PROGRAM MAIN
VAR
	brun 		AT %Q* : BOOL;
	bACK 		AT %Q* : BOOL;
	bSafety_OK  AT %I* : BOOL;
	bInit              : BOOL;
	Initialize		   : R_TRIG;
	Ack_Input		   : BOOL;
	Safety_Timer       : TON;	
	SafeOP_Timer	   : TON;
	EMG_Raise		   : R_TRIG;
	OP10A_Robo_State AT %I* : USINT;
	OP10B_Robo_State AT %I* : USINT;

	SERVO_TORQUE	AT %Q*	:UINT := 10000;
	
	ALL_LIGHTS_ON: BOOL;
	XTS_Lube_ON  : BOOL;
	
	All_Station_Auto_Mode     : BOOL;
	All_Station_Cycle_Start   : BOOL;
	All_Station_Cycle_Stop    : BOOL;
	Station_Ctrl_Temp         : BOOL;
	OP10_Lights_On			  : BOOL;
	tower_lamp_green_on       :BOOL;
	tower_lamp_red_on         :BOOL;
	tower_lamp_orange_on: BOOL;
	
	FB_Timer : FB_Time_Stamp_Maddy;
	Run_Time : STRING;
	Start_timer : BOOL;
	Stop_timer  : BOOL;
	Reset_timer : BOOL;
	Start_value : STRING;
	Stop_value  : STRING;
	Start_trig : R_TRIG;
	Stop_Trig  : R_TRIG;
	Reset_Trig : R_TRIG;
END_VAR


bACK			:= Pulse_Block.Q1Hz;

//Axis_Position_Bias();
O160_AUTOBAG_CNT_CMPLTD_Q707_4:=I10A_DRUM_OFF_ON_I714_2;
Initialize(CLK:=NOT bInit);
IF Initialize.Q THEN
	Ack_Input:=1;
	brun:=TRUE;
END_IF
SafeOP_Timer(IN:=Ack_Input,PT:=T#5S);
IF SafeOP_Timer.Q THEN
 bACK:=TRUE;
 Ack_Input:=0;
 bInit:=TRUE;
END_IF

Safety_Timer(IN:=bACK,PT:=T#500MS);
IF Safety_Timer.Q THEN
	bACK:=FALSE;
END_IF

EMG_Raise(CLK:=bSafety_OK , Q=> );
IF EMG_Raise.Q THEN
   bACK:=TRUE;
END_IF

RFID();
Error();
OP10_MAIN();
OP20_MAIN();
OP30_MAIN();
OP40_MAIN();
OP50_MAIN();
OP60_MAIN();
OP70_MAIN();
OP80_MAIN();
OP90_MAIN();
OP110_MAIN();
OP120_MAIN();
OP130_MAIN();
OP140_MAIN();
OP160_MAIN();
IO_Diag();
IO_OP10_PANEL();
IO_OP10A_10B_JB();
Master1_IO_Map();
MASTER2_IO_Map();
OP90_MP_IO();
OP90_MASTER3_IO();
OP90_JB_IO();
OP160_MP_IO();
OP160_MASTER4_IO();
OP120_JB_IO();
OP150_Main();
MAIN_1();
EtherCatDiag();
//MOdeselection From HMI
IF (HMI_AutoMode AND NOT HMI_ManualMOde AND NOT HMI_StepMode) THEN
		FB_MODE_BLOCK.ModeWord:=1;
	ELSIF (NOT HMI_AutoMode AND HMI_ManualMOde AND NOT HMI_StepMode) THEN
		FB_MODE_BLOCK.ModeWord:=2;
	ELSIF  (NOT HMI_AutoMode AND NOT HMI_ManualMOde AND HMI_StepMode) THEN
		FB_MODE_BLOCK.ModeWord:=3;
    ELSE   
		FB_MODE_BLOCK.ModeWord:=0;
END_IF

Servo_safety     := bSafety_OK;
OperationEnable  := bSafety_OK;

IF OperationEnable THEN
	Servo_Enable:=TRUE;
ELSE
	Servo_Enable:=FALSE;
END_IF

FB_MODE_BLOCK(
	ModeWord:= , 
	HomeConditionOK:= ALL_STN_IN_HOME, 
	OperationEnable:= bSafety_OK , 
	StartPB:= START_PB, 
	SafetyAndNOError:= bSafety_OK AND NOT ERROR_ACTIVE, 
	ModeAck:= TRUE , 
	HomingINProgress:= , 
	TempHomeOK:= , 
	ResetPB:= , 
	AutoSelected=>AUTO_SELECTED , 
	ManualSelected=> MANUAL_SELECTED, 
	StepSelected=> STEP_SELECTED, 
	ModeSelAck_Indication=> , 
	StatusDisplay=> , 
	AutoRunning:=AUTO_RUNNING , 
	StepRunning:=STEP_RUNNING , 
	StartEnable:=START_ENABLE , 
	MachineStop:=MACHINE_STOP);
	
Pulse_Block(
	Q10Hz=> , 
	Q5Hz=> , 
	Q2_5Hz=> , 
	Q2Hz=> , 
	Q1_25Hz=> , 
	Q2Hz=> , 
	Q0_625Hz=> , 
	Q0_5Hz=> );	
	
IF ALL_LIGHTS_ON THEN				
		O30_CAM_LGHT1_ON_Q305_1                  :=1;
		O30_CAM_LGHT2_ON_Q305_2                  :=1;
		O50_CAM_LGHT1_ON_Q306_3                  :=1;
		O50_CAM_LGHT2_ON_Q306_4                  :=1;
		O70_CAM_LGHT1_ON_Q307_6                  :=1;
		O70_CAM_LGHT2_ON_Q307_7                  :=1;
		O90_VISN_LGHT1_ON_Q400_0                 :=1;
		O90_VISN_LGHT2_ON_Q400_1                 :=1;
		O120_VISN_LGHT1_ON_Q402_4                :=1;
		O120_VISN_LGHT2_ON_Q402_5                :=1;
		O150_VISN_LGHT_ON_Q706_6                 :=1;
		O160_CHECKER_LGHT_ON_Q707_1              :=1;
ELSE		
		O30_CAM_LGHT1_ON_Q305_1                  :=0;
		O30_CAM_LGHT2_ON_Q305_2                  :=0;
		O50_CAM_LGHT1_ON_Q306_3                  :=0;
		O50_CAM_LGHT2_ON_Q306_4                  :=0;
		O70_CAM_LGHT1_ON_Q307_6                  :=0;
		O70_CAM_LGHT2_ON_Q307_7                  :=0;
		O90_VISN_LGHT1_ON_Q400_0                 :=0;
		O90_VISN_LGHT2_ON_Q400_1                 :=0;
		O120_VISN_LGHT1_ON_Q402_4                :=0;
		O120_VISN_LGHT2_ON_Q402_5                :=0;
		O150_VISN_LGHT_ON_Q706_6                 :=0;
		O160_CHECKER_LGHT_ON_Q707_1              :=0;	
END_IF

IF OP10_Lights_On THEN
		O10A_BDY_EMPT_CAM_LGHT1_ON_Q301_0        :=1; 
		O10A_BDY_EMPT_CAM_LGHT2_ON_Q301_1        :=1;
//		O10A_FIRTREE_ORING_CAM_LGHT1_ON_Q301_2   :=1;
//		O10A_FIRTREE_ORING_CAM_LGHT2_ON_Q301_3   :=1;
		O10A_ORING_CAM_LGHT1_ON_Q301_4           :=1;
		O10A_ORING_CAM_LGHT2_ON_Q301_5           :=1;
//		O10A_FIRTREE_ORING_CAMBAR_LGHT1_ON_Q301_6:=1;
//		O10B_FIRTREE_ORING_CAM_LGHT1_ON_Q303_2   :=1;
//		O10B_FIRTREE_ORING_CAM_LGHT2_ON_Q303_3   :=1;
		O10B_ORING_CAM_LGHT1_ON_Q303_4           :=1;
		O10B_ORING_CAM_LGHT2_ON_Q303_5           :=1;
//		O10B_FIRTREE_ORING_CAMBAR_LGHT1_ON_Q303_6:=1;
ELSE
		O10A_BDY_EMPT_CAM_LGHT1_ON_Q301_0        :=0; 
		O10A_BDY_EMPT_CAM_LGHT2_ON_Q301_1        :=0;
		O10A_FIRTREE_ORING_CAM_LGHT1_ON_Q301_2   :=0;
		O10A_FIRTREE_ORING_CAM_LGHT2_ON_Q301_3   :=0;
		O10A_ORING_CAM_LGHT1_ON_Q301_4           :=0;
		O10A_ORING_CAM_LGHT2_ON_Q301_5           :=0;
		O10A_FIRTREE_ORING_CAMBAR_LGHT1_ON_Q301_6:=0;
		O10B_FIRTREE_ORING_CAM_LGHT1_ON_Q303_2   :=0;
		O10B_FIRTREE_ORING_CAM_LGHT2_ON_Q303_3   :=0;
		O10B_ORING_CAM_LGHT1_ON_Q303_4           :=0;
		O10B_ORING_CAM_LGHT2_ON_Q303_5           :=0;
		O10B_FIRTREE_ORING_CAMBAR_LGHT1_ON_Q303_6:=0;	
END_IF
		
		
IF XTS_Lube_ON THEN
	O10_XTS_GREASE_VALVE_ON_Q300_0:=Pulse_Block.Q0_5Hz;
ELSE	
	O10_XTS_GREASE_VALVE_ON_Q300_0:=0;
END_IF
		
O150_BARLIGHT_OP1_Q706_7 :=	Pulse_Block.Q2_5Hz;
O150_BARLIGHT_OP2_Q707_0 := Pulse_Block.Q1Hz;	
                                                      
O10_TWR_LMP_RD_Q302_5   := Pulse_Block.Q1Hz AND tower_lamp_green_on;                         
O10_TWR_LMP_GN_Q302_6   := Pulse_Block.Q1Hz AND tower_lamp_red_on;                        
O10_TWR_LMP_YELW_Q302_7 := Pulse_Block.Q1Hz AND tower_lamp_orange_on;
O120_TWR_LMP_GN_Q403_1   := Pulse_Block.Q1Hz AND tower_lamp_green_on;
O120_TWR_LMP_YELW_Q403_2 := Pulse_Block.Q1Hz AND tower_lamp_orange_on ;
O120_TWR_LMP_RD_Q403_0   := Pulse_Block.Q1Hz AND tower_lamp_red_on;	

O10_BARLIGHT_OP1_Q300_6  := Pulse_Block.Q1Hz;
O10_BARLIGHT_OP2_Q300_7  := Pulse_Block.Q1_25Hz;	

IF NOT OperationEnable THEN
	OP20_ErrorActive:=1;
	OP30_ErrorActive:=1;
	OP40_ErrorActive:=1;
	OP50_ErrorActive:=1;
	OP60_ErrorActive:=1;
	OP70_ErrorActive:=1;
	OP80_ErrorActive:=1;
	OP110_ErrorActive:=1;
	OP120_ErrorActive:=1;
	OP130_ErrorActive:=1;
	OP140_ErrorActive:=1;
	OP160_ErrorActive:=1;
END_IF

IF AUTO_WITH_XTS AND Station_Ctrl_Temp THEN

	IF All_Station_Auto_Mode THEN
		OP20_HMI_AutoMode:=1;
		OP30_HMI_AutoMode:=1;
		OP40_HMI_AutoMode:=1;
		OP50_HMI_AutoMode:=1;
		OP60_HMI_AutoMode:=1;
		OP70_HMI_AutoMode:=1;
		OP80_HMI_AutoMode:=1;	
		OP110_HMI_AutoMode:=1;	
        OP120_HMI_AutoMode:=1;
		OP130_HMI_AutoMode:=1;	
	//	OP140_HMI_AutoMode:=1;
        OP160_HMI_AutoMode:=1;			
	END_IF
	IF All_Station_Cycle_Start THEN
		OP20_HMI_CycleStart	:=1;
		OP30_HMI_Cycle_Start:=1;
		OP40_HMI_Cycle_Start:=1;
		OP50_HMI_Cycle_Start:=1;
		OP60_HMI_CycleStart	:=1;
		OP70_HMI_Cycle_Start:=1;
		OP80_HMI_CycleStart	:=1;
		OP110_HMI_CycleStart:=1;
		OP120_HMI_CycleStart_PB:=1;
		OP130_HMI_CycleStart:=1;
	//	OP140_HMI_CycleStart:=1;
		OP160_HMI_CycleStart:=1;
	ELSE
		OP20_HMI_CycleStart	:=0;
		OP30_HMI_Cycle_Start:=0;
		OP40_HMI_Cycle_Start:=0;
		OP50_HMI_Cycle_Start:=0;
		OP60_HMI_CycleStart	:=0;
		OP70_HMI_Cycle_Start:=0;
		OP80_HMI_CycleStart	:=0;
		OP110_HMI_CycleStart:=0;	
		OP120_HMI_CycleStart_PB:=0;
		OP130_HMI_CycleStart:=0;
	//	OP140_HMI_CycleStart:=0;
		OP160_HMI_CycleStart:=0;		
	END_IF
	IF All_Station_Cycle_Stop THEN
		 OP20_Stop_Request  :=1;
 		 OP30_Stop_Request  :=1;
 		 OP40_Stop_Request  :=1;
 		 OP50_Stop_Request  :=1;
 		 OP60_Stop_Request  :=1;
 		 OP70_Stop_Request  :=1;
 		 OP80_Stop_Request  :=1;
 		 OP110_Stop_Request :=1;
		 OP120_Machine_Stop :=1;
		 OP130_Machine_Stop	:=1;
		// OP140_Machine_Stop :=1;
		 OP160_Machine_Stop	:=1;
	ELSE
		 OP20_Stop_Request  :=0;
 		 OP30_Stop_Request  :=0;
 		 OP40_Stop_Request  :=0;
 		 OP50_Stop_Request  :=0;
 		 OP60_Stop_Request  :=0;
 		 OP70_Stop_Request  :=0;
 		 OP80_Stop_Request  :=0;
 		 OP110_Stop_Request :=0;
		 OP120_Machine_Stop :=0;
		 OP130_Machine_Stop	:=0;
		// OP140_Machine_Stop :=0;
		 OP160_Machine_Stop	:=0;	 
	END_IF
END_IF	


////// tower lamp ////////////////////
IF OP10A_AUTO_RUNNING AND  OP160_AutoRunning AND  OP140_AutoRunning AND 
   OP130_AutoRunning AND OP110_AutoRunning AND OP120_AutoRunning  AND 
   OP90_AUTO_RUNNING AND OP80_AutoRunning AND OP70_AutoRunning AND 
   OP60_AutoRunning AND  OP50_AutoRunning AND OP40_AutoRunning AND 
   OP30_AutoRunning AND OP20_AutoRunning THEN
   tower_lamp_green_on := TRUE;
   tower_lamp_red_on   := FALSE;
   tower_lamp_orange_on:=FALSE;	
END_IF

IF NOT (OP160_AutoRunning AND  OP140_AutoRunning AND  OP130_AutoRunning AND 
        OP10A_AUTO_RUNNING AND OP110_AutoRunning AND OP120_AutoRunning AND
        OP90_AUTO_RUNNING AND OP80_AutoRunning AND OP70_AutoRunning AND
        OP60_AutoRunning AND OP50_AutoRunning AND OP40_AutoRunning AND
        OP30_AutoRunning AND OP20_AutoRunning) THEN
	    tower_lamp_green_on :=FALSE ;
	    tower_lamp_red_on   := FALSE;
        tower_lamp_orange_on:=TRUE;	
END_IF

IF  OP10A_ERR OR OP10B_ERR OR OP110_ErrorActive OR OP120_ErrorActive OR OP130_ErrorActive OR OP140_ErrorActive
    OR OP160_ErrorActive OR OP90_ERR OR OP80_ErrorActive OR OP70_ErrorActive OR OP60_ErrorActive OR
	OP50_ErrorActive OR OP40_ErrorActive OR OP30_ErrorActive OR OP20_ErrorActive THEN
        tower_lamp_green_on :=FALSE ;
		tower_lamp_red_on   := TRUE;
		tower_lamp_orange_on:=FALSE;	
END_IF			
		
//////////////////

fbTime();

logTimer( IN := fbTime.bValid );
IF logTimer.Q THEN
    logTimer( IN := FALSE );
	logTimer( IN := fbTime.bValid );
    ADSLOGSTR( ADSLOG_MSGTYPE_HINT OR ADSLOG_MSGTYPE_LOG, 'Local System Time:%s', SYSTEMTIME_TO_STRING(fbTime.systemTime));
END_IF	

	wYear	:= fbTime.systemTime.wYear;
	wMonth	:= fbTime.systemTime.wMonth;
	wDate   := fbTime.systemTime.wDay;
	wHour	:= fbTime.systemTime.wHour;
	wMinute := fbTime.systemTime.wMinute;
	wSecond := fbTime.systemTime.wSecond;
	wMillisec:= fbTime.systemTime.wMilliseconds;
	
FB_Timer(
	Start:= , 
	Stop:= , 
	Running_Timer=> Run_Time, 
	Time_Difference_ms=> , 
	Time_Struct:=fbTime.systemTime );	
	
Start_trig(CLK:=Start_timer);	
Stop_trig(CLK :=Stop_timer);
Reset_Trig(CLK:=Reset_timer);	
	
IF Start_trig.Q THEN
	Start_value:=Run_Time;
END_IF
IF Stop_trig.Q THEN
	Stop_value:=Run_Time;
END_IF
IF Reset_Trig.Q THEN
	Start_value:=' ';
	Stop_value:=' ';
END_IF

END_PROGRAM

(* stored: Version 1.1.0.1, ProductVersion 3.1.4024.11
   POU MAIN: Id {fd835ba8-4538-4711-9017-05a7c6c2ed82}, SpecialFunc None *)
